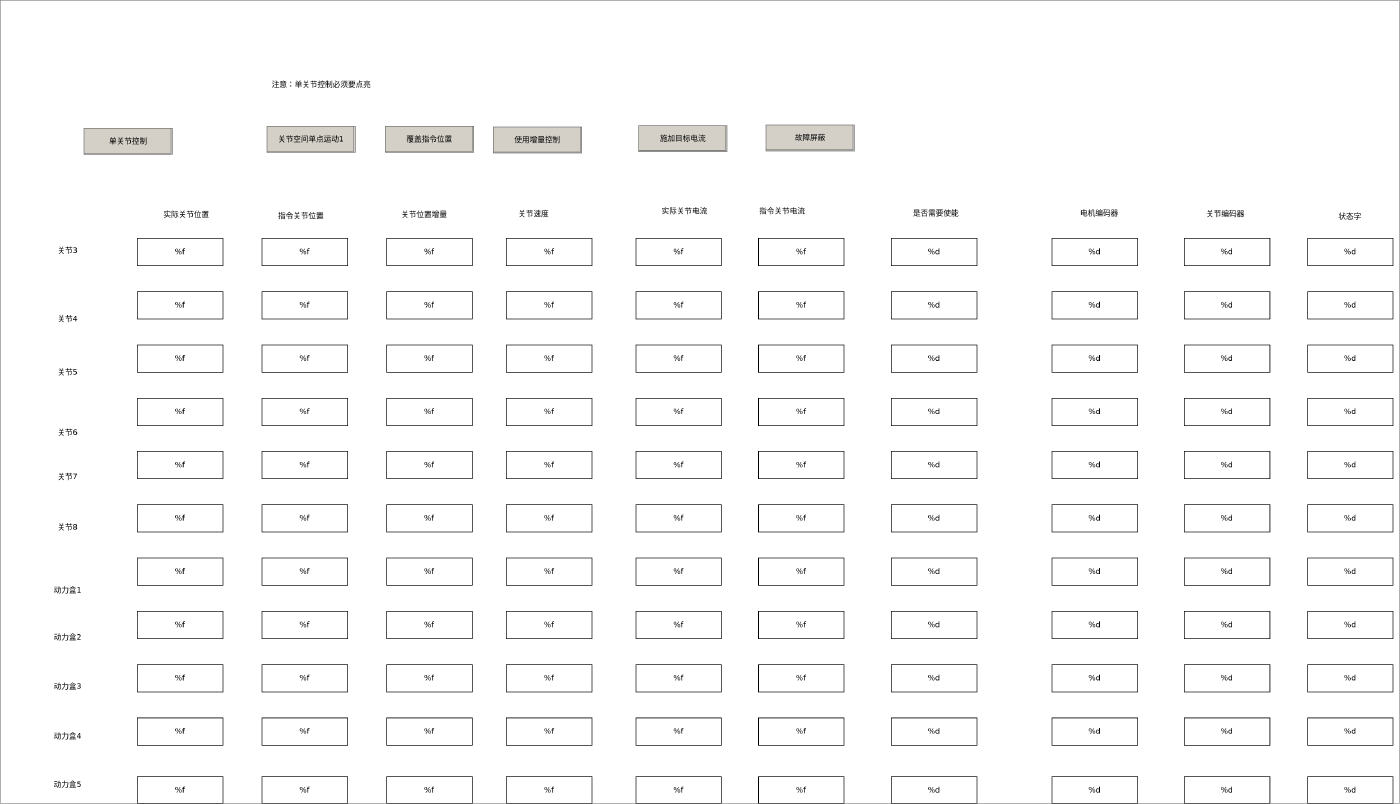
VISUALIZATION motion_a1  // 2022x1162
    Button (385,182 128x38), "关节空间单点运动1", colour toggle: g_motionTest.m_uiArmMode[1,1]
        tap g_motionTest.m_uiArmMode[1,1]
    Label (362,298 145x28), "指令关节位置"
    Label (194,295 150x30), "实际关节位置"
    Label (540,296 145x28), "关节位置增量"
    Label (698,295 145x28), "关节速度"
    Label (916,291 145x28), "实际关节电流"
    Label (1057,291 145x28), "指令关节电流"
    Rectangle (198,575 124x40), "%f", text variable: g_motionTest.m_actJntPos[1][1]
    Label (25,348 145x28), "关节3"
    Label (25,447 145x28), "关节4"
    Label (25,524 145x28), "关节5"
    Label (25,611 145x28), "关节6"
    Label (25,675 145x28), "关节7"
    Label (25,748 145x28), "关节8"
    Label (25,839 145x28), "动力盒1"
    Label (25,907 145x28), "动力盒2"
    Label (25,1120 145x28), "动力盒5"
    Label (25,978 145x28), "动力盒3"
    Label (25,1050 145x28), "动力盒4"
    Rectangle (198,652 124x40), "%f", text variable: g_motionTest.m_actJntPos[1][2]
    Rectangle (198,729 124x40), "%f", text variable: g_motionTest.m_actJntPos[1][3]
    Rectangle (198,806 124x40), "%f", text variable: g_motionTest.m_actJntPos[1][4]
    Rectangle (198,883 124x40), "%f", text variable: g_motionTest.m_actJntPos[1][5]
    Rectangle (198,960 124x40), "%f", text variable: g_motionTest.m_actJntPos[1][6]
    Rectangle (198,1037 124x40), "%f", text variable: g_motionTest.m_actJntPos[1][7]
    Rectangle (198,1122 124x40), "%f", text variable: g_motionTest.m_actJntPos[1][8]
    Rectangle (198,344 124x40), "%f", text variable: g_motionTest.m_actJntPosSetup[1][3]
    Rectangle (198,421 124x40), "%f", text variable: g_motionTest.m_actJntPosSetup[1][4]
    Rectangle (198,498 124x40), "%f", text variable: g_motionTest.m_actJntPosSetup[1][5]
    Rectangle (378,344 124x40), "%f", text variable: g_motionTest.m_targetJntPosSetup[1][3]
        OnMouseClick: write the text variable via Default
    Rectangle (378,421 124x40), "%f", text variable: g_motionTest.m_targetJntPosSetup[1][4]
        OnMouseClick: write the text variable via Default
    Rectangle (378,498 124x40), "%f", text variable: g_motionTest.m_targetJntPosSetup[1][5]
        OnMouseClick: write the text variable via Default
    Rectangle (378,575 124x40), "%f", text variable: g_motionTest.m_targetJntPosN8[1][1]
        OnMouseClick: write the text variable via Default
    Rectangle (378,652 124x40), "%f", text variable: g_motionTest.m_targetJntPosN8[1][2]
        OnMouseClick: write the text variable via Default
    Rectangle (378,729 124x40), "%f", text variable: g_motionTest.m_targetJntPosN8[1][3]
        OnMouseClick: write the text variable via Default
    Rectangle (378,806 124x40), "%f", text variable: g_motionTest.m_targetJntPosN8[1][4]
        OnMouseClick: write the text variable via Default
    Rectangle (378,883 124x40), "%f", text variable: g_motionTest.m_targetJntPosN8[1][5]
        OnMouseClick: write the text variable via Default
    Rectangle (378,960 124x40), "%f", text variable: g_motionTest.m_targetJntPosN8[1][6]
        OnMouseClick: write the text variable via Default
    Rectangle (378,1037 124x40), "%f", text variable: g_motionTest.m_targetJntPosN8[1][7]
        OnMouseClick: write the text variable via Default
    Rectangle (378,1122 124x40), "%f", text variable: g_motionTest.m_targetJntPosN8[1][8]
        OnMouseClick: write the text variable via Default
    Rectangle (558,344 124x40), "%f", text variable: g_motionTest.m_targetJntPosIncSetup[1][3]
        OnMouseClick: write the text variable via Default
    Rectangle (558,421 124x40), "%f", text variable: g_motionTest.m_targetJntPosIncSetup[1][4]
        OnMouseClick: write the text variable via Default
    Rectangle (558,498 124x40), "%f", text variable: g_motionTest.m_targetJntPosIncSetup[1][5]
        OnMouseClick: write the text variable via Default
    Rectangle (558,575 124x40), "%f", text variable: g_motionTest.m_targetJntPosIncN8[1][1]
        OnMouseClick: write the text variable via Default
    Rectangle (558,652 124x40), "%f", text variable: g_motionTest.m_targetJntPosIncN8[1][2]
        OnMouseClick: write the text variable via Default
    Rectangle (558,729 124x40), "%f", text variable: g_motionTest.m_targetJntPosIncN8[1][3]
        OnMouseClick: write the text variable via Default
    Rectangle (558,806 124x40), "%f", text variable: g_motionTest.m_targetJntPosIncN8[1][4]
        OnMouseClick: write the text variable via Default
    Rectangle (558,883 124x40), "%f", text variable: g_motionTest.m_targetJntPosIncN8[1][5]
        OnMouseClick: write the text variable via Default
    Rectangle (558,960 124x40), "%f", text variable: g_motionTest.m_targetJntPosIncN8[1][6]
        OnMouseClick: write the text variable via Default
    Rectangle (558,1037 124x40), "%f", text variable: g_motionTest.m_targetJntPosIncN8[1][7]
        OnMouseClick: write the text variable via Default
    Rectangle (558,1122 124x40), "%f", text variable: g_motionTest.m_targetJntPosIncN8[1][8]
        OnMouseClick: write the text variable via Default
    Rectangle (731,344 124x40), "%f", text variable: g_motionTest.m_targetJntVelSetup[1][3]
        OnMouseClick: write the text variable via Default
    Rectangle (731,421 124x40), "%f", text variable: g_motionTest.m_targetJntVelSetup[1][4]
        OnMouseClick: write the text variable via Default
    Rectangle (731,498 124x40), "%f", text variable: g_motionTest.m_targetJntVelSetup[1][5]
        OnMouseClick: write the text variable via Default
    Rectangle (731,575 124x40), "%f", text variable: g_motionTest.m_targetJntVel[1][1]
        OnMouseClick: write the text variable via Default
    Rectangle (731,652 124x40), "%f", text variable: g_motionTest.m_targetJntVel[1][2]
        OnMouseClick: write the text variable via Default
    Rectangle (731,729 124x40), "%f", text variable: g_motionTest.m_targetJntVel[1][3]
        OnMouseClick: write the text variable via Default
    Rectangle (731,806 124x40), "%f", text variable: g_motionTest.m_targetJntVel[1][4]
        OnMouseClick: write the text variable via Default
    Rectangle (731,883 124x40), "%f", text variable: g_motionTest.m_targetJntVel[1][5]
        OnMouseClick: write the text variable via Default
    Rectangle (731,960 124x40), "%f", text variable: g_motionTest.m_targetJntVel[1][6]
        OnMouseClick: write the text variable via Default
    Rectangle (731,1037 124x40), "%f", text variable: g_motionTest.m_targetJntVel[1][7]
        OnMouseClick: write the text variable via Default
    Rectangle (731,1122 124x40), "%f", text variable: g_motionTest.m_targetJntVel[1][8]
        OnMouseClick: write the text variable via Default
    Rectangle (918,344 124x40), "%f", text variable: g_motionTest.m_actJntCurrentSetup[1][3]
    Rectangle (918,421 124x40), "%f", text variable: g_motionTest.m_actJntCurrentSetup[1][4]
    Rectangle (918,498 124x40), "%f", text variable: g_motionTest.m_actJntCurrentSetup[1][5]
    Rectangle (918,575 124x40), "%f", text variable: g_motionTest.m_actJntCurrent[1][1]
    Rectangle (918,652 124x40), "%f", text variable: g_motionTest.m_actJntCurrent[1][2]
    Rectangle (918,729 124x40), "%f", text variable: g_motionTest.m_actJntCurrent[1][3]
    Rectangle (918,806 124x40), "%f", text variable: g_motionTest.m_actJntCurrent[1][4]
    Rectangle (918,883 124x40), "%f", text variable: g_motionTest.m_actJntCurrent[1][5]
    Rectangle (918,960 124x40), "%f", text variable: g_motionTest.m_actJntCurrent[1][6]
    Rectangle (918,1037 124x40), "%f", text variable: g_motionTest.m_actJntCurrent[1][7]
    Rectangle (918,1122 124x40), "%f", text variable: g_motionTest.m_actJntCurrent[1][8]
    Rectangle (1095,344 124x40), "%f", text variable: g_motionTest.m_targetJntCurrentSetup[1][3]
        OnMouseClick: write the text variable via Default
    Rectangle (1095,421 124x40), "%f", text variable: g_motionTest.m_targetJntCurrentSetup[1][4]
        OnMouseClick: write the text variable via Default
    Rectangle (1095,498 124x40), "%f", text variable: g_motionTest.m_targetJntCurrentSetup[1][5]
        OnMouseClick: write the text variable via Default
    Rectangle (1095,575 124x40), "%f", text variable: g_motionTest.m_targetJntCurrentN8[1][1]
        OnMouseClick: write the text variable via Default
    Rectangle (1095,652 124x40), "%f", text variable: g_motionTest.m_targetJntCurrentN8[1][2]
        OnMouseClick: write the text variable via Default
    Rectangle (1095,729 124x40), "%f", text variable: g_motionTest.m_targetJntCurrentN8[1][3]
        OnMouseClick: write the text variable via Default
    Rectangle (1095,806 124x40), "%f", text variable: g_motionTest.m_targetJntCurrentN8[1][4]
        OnMouseClick: write the text variable via Default
    Rectangle (1095,883 124x40), "%f", text variable: g_motionTest.m_targetJntCurrentN8[1][5]
        OnMouseClick: write the text variable via Default
    Rectangle (1095,960 124x40), "%f", text variable: g_motionTest.m_targetJntCurrentN8[1][6]
        OnMouseClick: write the text variable via Default
    Rectangle (1095,1037 124x40), "%f", text variable: g_motionTest.m_targetJntCurrentN8[1][7]
        OnMouseClick: write the text variable via Default
    Rectangle (1095,1122 124x40), "%f", text variable: g_motionTest.m_targetJntCurrentN8[1][8]
        OnMouseClick: write the text variable via Default
    Button (712,183 128x38), "使用增量控制", colour toggle: g_motionTest.m_singleMotorIncControl[1]
        toggle g_motionTest.m_singleMotorIncControl[1]
    Button (922,181 128x38), "施加目标电流", colour toggle: g_motionTest.m_uiArmMode[1,9]
        toggle g_motionTest.m_uiArmMode[1,9]
    Button (121,185 128x38), "单关节控制", colour toggle: g_motionTest.m_singleMotorControl[1]
        toggle g_motionTest.m_singleMotorControl[1]
    Label (354,107 220x30), "注意：单关节控制必须要点亮"
    Label (1279,293 145x30), "是否需要使能"
    Rectangle (1287,344 124x40), "%d", text variable: g_motionTest.m_jntEnableSetup[1][3]
        OnMouseClick: write the text variable via Default
    Rectangle (1287,421 124x40), "%d", text variable: g_motionTest.m_jntEnableSetup[1][4]
        OnMouseClick: write the text variable via Default
    Rectangle (1287,498 124x40), "%d", text variable: g_motionTest.m_jntEnableSetup[1][5]
        OnMouseClick: write the text variable via Default
    Rectangle (1287,575 124x40), "%d", text variable: g_motionTest.m_jntEnable[1][1]
        OnMouseClick: write the text variable via Default
    Rectangle (1287,652 124x40), "%d", text variable: g_motionTest.m_jntEnable[1][2]
        OnMouseClick: write the text variable via Default
    Rectangle (1287,729 124x40), "%d", text variable: g_motionTest.m_jntEnable[1][3]
        OnMouseClick: write the text variable via Default
    Rectangle (1287,806 124x40), "%d", text variable: g_motionTest.m_jntEnable[1][4]
        OnMouseClick: write the text variable via Default
    Rectangle (1287,883 124x40), "%d", text variable: g_motionTest.m_jntEnable[1][5]
        OnMouseClick: write the text variable via Default
    Rectangle (1287,960 124x40), "%d", text variable: g_motionTest.m_jntEnable[1][6]
        OnMouseClick: write the text variable via Default
    Rectangle (1287,1037 124x40), "%d", text variable: g_motionTest.m_jntEnable[1][7]
        OnMouseClick: write the text variable via Default
    Rectangle (1287,1122 124x40), "%d", text variable: g_motionTest.m_jntEnable[1][8]
        OnMouseClick: write the text variable via Default
    Label (1515,294 145x28), "电机编码器"
    Label (1697,295 145x28), "关节编码器"
    Label (1877,299 145x28), "状态字"
    Rectangle (1519,344 124x40), "%d", text variable: g_systemInfo.m_setupJntInfo[1,3].m_motorInput.m_motorEncoder
    Rectangle (1519,421 124x40), "%d", text variable: g_systemInfo.m_setupJntInfo[1,4].m_motorInput.m_motorEncoder
    Rectangle (1519,498 124x40), "%d", text variable: g_systemInfo.m_setupJntInfo[1,5].m_motorInput.m_motorEncoder
    Rectangle (1519,575 124x40), "%d", text variable: g_systemInfo.m_slaveJntInfo[1,1].m_motorInput.m_motorEncoder
    Rectangle (1519,652 124x40), "%d", text variable: g_systemInfo.m_slaveJntInfo[1,2].m_motorInput.m_motorEncoder
    Rectangle (1519,729 124x40), "%d", text variable: g_systemInfo.m_slaveJntInfo[1,3].m_motorInput.m_motorEncoder
    Rectangle (1519,806 124x40), "%d", text variable: g_systemInfo.m_slaveJntInfo[1,4].m_motorInput.m_motorEncoder
    Rectangle (1519,883 124x40), "%d", text variable: g_systemInfo.m_slaveJntInfo[1,5].m_motorInput.m_motorEncoder
    Rectangle (1519,960 124x40), "%d", text variable: g_systemInfo.m_slaveJntInfo[1,6].m_motorInput.m_motorEncoder
    Rectangle (1519,1037 124x40), "%d", text variable: g_systemInfo.m_slaveJntInfo[1,7].m_motorInput.m_motorEncoder
    Rectangle (1519,1122 124x40), "%d", text variable: g_systemInfo.m_slaveJntInfo[1,8].m_motorInput.m_motorEncoder
    Rectangle (1710,344 124x40), "%d", text variable: g_systemInfo.m_setupJntInfo[1,3].m_motorInput.m_linkEncoder
    Rectangle (1710,421 124x40), "%d", text variable: g_systemInfo.m_setupJntInfo[1,4].m_motorInput.m_linkEncoder
    Rectangle (1710,498 124x40), "%d", text variable: g_systemInfo.m_setupJntInfo[1,5].m_motorInput.m_linkEncoder
    Rectangle (1710,575 124x40), "%d", text variable: g_systemInfo.m_slaveJntInfo[1,1].m_motorInput.m_linkEncoder
    Rectangle (1710,652 124x40), "%d", text variable: g_systemInfo.m_slaveJntInfo[1,2].m_motorInput.m_linkEncoder
    Rectangle (1710,729 124x40), "%d", text variable: g_systemInfo.m_slaveJntInfo[1,3].m_motorInput.m_linkEncoder
    Rectangle (1710,806 124x40), "%d", text variable: g_systemInfo.m_slaveJntInfo[1,4].m_motorInput.m_linkEncoder
    Rectangle (1710,883 124x40), "%d", text variable: g_systemInfo.m_slaveJntInfo[1,5].m_motorInput.m_linkEncoder
    Rectangle (1710,960 124x40), "%d", text variable: g_systemInfo.m_slaveJntInfo[1,6].m_motorInput.m_linkEncoder
    Rectangle (1710,1037 124x40), "%d", text variable: g_systemInfo.m_slaveJntInfo[1,7].m_motorInput.m_linkEncoder
    Rectangle (1710,1122 124x40), "%d", text variable: g_systemInfo.m_slaveJntInfo[1,8].m_motorInput.m_linkEncoder
    Rectangle (1888,344 124x40), "%d", text variable: g_systemInfo.m_setupJntInfo[1,3].m_motorInput.m_statusWord
    Rectangle (1888,421 124x40), "%d", text variable: g_systemInfo.m_setupJntInfo[1,4].m_motorInput.m_statusWord
    Rectangle (1888,498 124x40), "%d", text variable: g_systemInfo.m_setupJntInfo[1,5].m_motorInput.m_statusWord
    Rectangle (1888,575 124x40), "%d", text variable: g_systemInfo.m_slaveJntInfo[1,1].m_motorInput.m_statusWord
    Rectangle (1888,652 124x40), "%d", text variable: g_systemInfo.m_slaveJntInfo[1,2].m_motorInput.m_statusWord
    Rectangle (1888,729 124x40), "%d", text variable: g_systemInfo.m_slaveJntInfo[1,3].m_motorInput.m_statusWord
    Rectangle (1888,806 124x40), "%d", text variable: g_systemInfo.m_slaveJntInfo[1,4].m_motorInput.m_statusWord
    Rectangle (1888,883 124x40), "%d", text variable: g_systemInfo.m_slaveJntInfo[1,5].m_motorInput.m_statusWord
    Rectangle (1888,960 124x40), "%d", text variable: g_systemInfo.m_slaveJntInfo[1,6].m_motorInput.m_statusWord
    Rectangle (1888,1037 124x40), "%d", text variable: g_systemInfo.m_slaveJntInfo[1,7].m_motorInput.m_statusWord
    Rectangle (1888,1122 124x40), "%d", text variable: g_systemInfo.m_slaveJntInfo[1,8].m_motorInput.m_statusWord
    Button (1106,180 128x38), "故障屏蔽", colour toggle: g_specialSignal.m_faultMask
        toggle g_specialSignal.m_faultMask
    Button (556,182 128x38), "覆盖指令位置", colour toggle: g_motionTest.m_coverCmdPos[1]
        tap g_motionTest.m_coverCmdPos[1]
END_VISUALIZATION

(* stored: Version 1.1.0.1, ProductVersion 3.1.4024.11
   Visu motion_a1: Id {8351ce4d-5a5a-4ccc-a562-c70180566038} *)
